TYPE ST_AxisError:
STRUCT
//PLCopen function block errors
    nPowerErrorID : UDINT;
    nMoveAbsoluteErrorID : UDINT;
    nMoveRelativeErrorID : UDINT;
    nMoveVelocityErrorID : UDINT;
    nMoveModuloErrorID : UDINT;
    nJogErrorID : UDINT;
    nHomeErrorID : UDINT;
    nHaltErrorID : UDINT;
    nResetErrorID : UDINT;
    nStopErrorID : UDINT;
    nGearInErrorID : UDINT;
    nGearInMultiMasterErrorID : UDINT;
    nGearOutErrorID : UDINT;
    fbWriteParameterErrorId : UDINT;
    fbReadParameterErrorId : UDINT;
//Error from the NC
    nNCErrorID : UDINT;
END_STRUCT
END_TYPE

(* stored: Version 1.1.0.1, ProductVersion 3.1.4024.11
   DUT ST_AxisError: Id {b605e536-99a4-4241-8b01-b55c227dfd1d} *)
